/// The state profile for position, velocity, acceleration and jerk for a single DoF
FUNCTION_BLOCK Profile
VAR_INPUT
  limits : ProfileLimitsEnum;
  direction : ProfileDirectionEnum;
  jerkSigns : ProfileJerkSignsEnum;
  
  t, t_sum, j : ARRAY[0..6] OF LREAL;
  a, v, p : ARRAY[0..7] OF LREAL;

  pf, vf, af : LREAL; // Target (final) kinematic state
  
  hasBrake : BOOL;
  t_brake : LREAL; // Total time of the braking segments
  t_brakes, j_brakes, a_brakes, v_brakes, p_brakes : ARRAY[0..1] OF LREAL; // Allow up to two segments of braking before the "correct" profile starts 

END_VAR
VAR CONSTANT
  eps : LREAL := 1E-8;  
  infinity : LREAL := 1.7976931348623157E+308;
END_VAR
VAR_STAT
  root : Roots;
END_VAR

METHOD check : BOOL
VAR_INPUT
  jerkSigns : ProfileJerkSignsEnum;    
  limits : ProfileLimitsEnum;
  tf : LREAL;
  jf : LREAL;
  vMax : LREAL;
  vMin : LREAL;  
  aMax : LREAL;
  aMin : LREAL;
  jMax  : LREAL;
END_VAR
check := (ABS(jf) < ABS(jMax) + 1e-12) AND_THEN checkTime(jerkSigns, limits, tf, jf, vMax, vMin, aMax, aMin);
END_METHOD

/// For velocity interface
METHOD checkAcc : BOOL
VAR_INPUT
  jerkSigns : ProfileJerkSignsEnum;
  limits : ProfileLimitsEnum;  
  jf : LREAL;
  aMax : LREAL;
  aMin : LREAL;  
END_VAR
VAR
  i : INT;
  aUppLim : LREAL;
  aLowLim : LREAL;
END_VAR
IF (t[0] < 0)
THEN
  RETURN;
END_IF

t_sum[0] := t[0];
FOR i:=0 TO 5
DO
  IF (t[i+1] < 0)
  THEN
    RETURN;
  END_IF
  
  t_sum[i+1] := t_sum[i] + t[i+1];
END_FOR


IF limits = ProfileLimitsEnum.acc0
THEN
  IF t[1] < eps
  THEN
    RETURN;
  END_IF
END_IF


IF (t_sum[6] > 1E12) { // For numerical reasons, is that needed?}
THEN
  RETURN;        
END_IF

IF jerkSigns = ProfileJerkSignsEnum.uddu
THEN
  j[0] := jf;
  j[1] := 0;
  j[2] := -jf;
  j[3] := 0;
  j[4] := -jf;
  j[5] := 0;
  j[6] := jf;          
ELSE
  j[0] := jf;
  j[1] := 0;
  j[2] := -jf;
  j[3] := 0;
  j[4] := jf;
  j[5] := 0;
  j[6] := -jf;
END_IF


FOR i:=0 TO 6
DO
  a[i+1] := a[i] + t[i] * j[i];
  v[i+1] := v[i] + t[i] * (a[i] + t[i] * j[i] / 2);
  p[i+1] := p[i] + t[i] * (v[i] + t[i] * (a[i] / 2 + t[i] * j[i] / 6));        
END_FOR

      
THIS^.jerkSigns := jerkSigns;
THIS^.limits := limits;

aUppLim := SEL((aMax > 0), aMin, aMax) + 1E-12;
aLowLim := SEL((aMax > 0), aMax, aMin) - 1E-12;

// Velocity limit can be broken in the beginning if both initial velocity and acceleration are too high
checkAcc := ABS(v[7] - vf) < 1E-8
    AND_THEN ABS(a[7] - af) < 1E-12 // This is not really needed, but we want to double check
    AND_THEN a[1] >= aLowLim AND_THEN a[3] >= aLowLim AND_THEN a[5] >= aLowLim
    AND_THEN a[1] <= aUppLim AND_THEN a[3] <= aUppLim AND_THEN a[5] <= aUppLim;
END_METHOD

METHOD checkPositionExtremum : BOOL
VAR_INPUT
  t_ext, t_sum, t, p, v, a, j : LREAL;
END_VAR
VAR_IN_OUT
  ext : PositionExtremaStruct;     
END_VAR
VAR
  p_ext, v_Ext, a_ext : LREAL;
END_VAR
IF (0 < t_ext AND_THEN t_ext < t)
THEN
  integrate(t_ext, p, v, a, j, p:=p_ext, v:=v_ext, a:=a_ext);
  IF (a_ext > 0 AND_THEN p_ext < ext.minimum)
  THEN
    ext.minimum := p_ext;
    ext.t_min := t_sum + t_ext;
   ELSIF (a_ext < 0 AND_THEN p_ext > ext.maximum) 
   THEN
    ext.maximum := p_ext;
    ext.t_max := t_sum + t_ext; 
  END_IF
END_IF
END_METHOD

METHOD checkStepForPositionExtremum : BOOL
VAR_INPUT
  t_sum, t, p, v, a, j : LREAL;
END_VAR
VAR_IN_OUT
  ext : PositionExtremaStruct;  
END_VAR
VAR
  d, d_sqrt : LREAL;
END_VAR
IF (p < ext.minimum)
THEN 
  ext.minimum := p;
  ext.t_min := t_sum;
END_IF

IF (p > ext.maximum)
THEN 
  ext.maximum := p;
  ext.t_max := t_sum;
END_IF

IF (j <> 0) 
THEN
  d := a * a - 2 * j * v;
  IF (ABS(d) < eps)
  THEN
    checkPositionExtremum(-a / j, t_sum, t, p, v, a, j, ext:=ext);
   ELSIF (d > 0) 
   THEN
    d_sqrt := SQRT(d);
    checkPositionExtremum((-a - D_sqrt) / j, t_sum, t, p, v, a, j, ext:=ext);
    checkPositionExtremum((-a + D_sqrt) / j, t_sum, t, p, v, a, j, ext:=ext);           
  END_IF
END_IF
END_METHOD

METHOD checkTime : BOOL
VAR_INPUT
  jerkSigns : ProfileJerkSignsEnum;    
  limits : ProfileLimitsEnum;
  tf : LREAL;
  jf : LREAL;
  vMax : LREAL;
  vMin : LREAL;  
  aMax : LREAL;
  aMin : LREAL;  
END_VAR
// Time doesn't need to be checked as every profile has a: tf - ... equation
checkTime := checkVel(jerkSigns, limits, jf, vMax, vMin, aMax, aMin); // && (std::abs(t_sum[6] - tf) < 1e-8)
END_METHOD

/// For position interface
METHOD checkVel : BOOL
VAR_INPUT
  jerkSigns : ProfileJerkSignsEnum;    
  limits : ProfileLimitsEnum;
  jf : LREAL;
  vMax : LREAL;
  vMin : LREAL;  
  aMax : LREAL;
  aMin : LREAL;
END_VAR
VAR
  i : INT;
  v_a_zero : LREAL;
  vUppLim, vLowLim : LREAL;  
  aUppLim, aLowLim : LREAL;
END_VAR
IF (t[0] < 0) 
THEN
  RETURN;
END_IF

t_sum[0] := t[0];
FOR i:=0 TO 5
DO
  IF (t[i+1] < 0)
  THEN
    RETURN;
  END_IF
  
  t_sum[i+1] := t_sum[i] + t[i+1];  
END_FOR

IF limits = ProfileLimitsEnum.acc0_acc1_vel OR_ELSE limits = ProfileLimitsEnum.acc0_vel OR_ELSE limits = ProfileLimitsEnum.acc1_vel OR_ELSE limits = ProfileLimitsEnum.vel
THEN
  IF (t[3] < eps) 
  THEN
    RETURN;                    
  END_IF
END_IF

IF limits = ProfileLimitsEnum.acc0 OR_ELSE limits = ProfileLimitsEnum.acc0_acc1
THEN
  IF (t[1] < eps) 
  THEN
    RETURN;                    
  END_IF
END_IF

IF limits = ProfileLimitsEnum.acc1 OR_ELSE limits = ProfileLimitsEnum.acc0_acc1
THEN
  IF (t[5] < eps)
  THEN
    RETURN;            
  END_IF
END_IF

IF t_sum[6] > 1E12  // For numerical reasons, is that needed?
THEN
  RETURN;        
END_IF
        
IF jerkSigns = ProfileJerkSignsEnum.uddu
THEN
  j[0] := jf;
  j[1] := 0;
  j[2] := -jf;
  j[3] := 0;
  j[4] := -jf;
  j[5] := 0;
  j[6] := jf;
ELSE
  j[0] := jf;
  j[1] := 0;
  j[2] := -jf;
  j[3] := 0;
  j[4] := jf;
  j[5] := 0;
  j[6] := -jf;          
END_IF

vUppLim := SEL(vMax > 0, vMin, vMax) + 1E-12;
vLowLim := SEL(vMax > 0, vMax, vMin) - 1E-12;
        
FOR i:= 0 TO 6 
DO
  a[i+1] := a[i] + t[i] * j[i];
  v[i+1] := v[i] + t[i] * (a[i] + t[i] * j[i] / 2);
  p[i+1] := p[i] + t[i] * (v[i] + t[i] * (a[i] / 2 + t[i] * j[i] / 6));

  IF limits = ProfileLimitsEnum.acc0_acc1_vel OR_ELSE limits = ProfileLimitsEnum.acc0_vel OR_ELSE limits = ProfileLimitsEnum.acc1_vel OR_ELSE limits = ProfileLimitsEnum.vel
  THEN
    IF i = 2
    THEN
     a[3] := 0.0;
    END_IF
  END_IF 
  
  IF (i > 1 AND_THEN a[i+1] * a[i] < -eps) 
  THEN
    v_a_zero := v[i] - (a[i] * a[i]) / (2 * j[i]);
    IF (v_a_zero > vUppLim OR_ELSE v_a_zero < vLowLim)
    THEN
      RETURN;        
		END_IF
  END_IF
END_FOR


THIS^.jerkSigns := jerkSigns;
THIS^.limits := limits;

aUppLim := SEL((aMax > 0), aMin, aMax) + 1E-12;
aLowLim := SEL((aMax > 0), aMax, aMin) - 1E-12;

// Velocity limit can be broken in the beginning if both initial velocity and acceleration are too high
checkVel := ABS(p[7] - pf) < 1E-8
    AND_THEN ABS(v[7] - vf) < 1E-8
    AND_THEN ABS(a[7] - af) < 1E-10 // This is not really needed, but we want to double check
    // AND_THEN ABS(v[3]) <= vMaxAbs AND_THEN ABS(v[4]) <= vMaxAbs AND_THEN ABS(v[5]) <= vMaxAbs AND_THEN ABS(v[6]) <= vMaxAbs
    AND_THEN a[1] >= aLowLim AND_THEN a[3] >= aLowLim AND_THEN a[5] >= aLowLim
    AND_THEN a[1] <= aUppLim AND_THEN a[3] <= aUppLim AND_THEN a[5] <= aUppLim
    AND_THEN v[3] <= vUppLim AND_THEN v[4] <= vUppLim AND_THEN v[5] <= vUppLim AND_THEN v[6] <= vUppLim
    AND_THEN v[3] >= vLowLim AND_THEN v[4] >= vLowLim AND_THEN v[5] >= vLowLim AND_THEN v[6] >= vLowLim; // this is not really needed, but we want to double check
END_METHOD

METHOD firstStateAtPosition : BOOL
VAR_INPUT
  pt, offset : LREAL;
END_VAR
VAR_IN_OUT
  t_t, v_t, a_t : LREAL;
END_VAR
VAR
  i,h : INT;
  p_t : LREAL;
  polynom : ARRAY[0..4] OF LREAL;
END_VAR
FOR i:=0 TO 6
DO
  IF ABS(p[i] - pt) < eps
  THEN
    t_t := offset + SEL(i>0, 0, t_sum[i-1]);
    v_t := v[i];
    a_t := a[i];
    firstStateAtPosition := TRUE;
    RETURN;
	END_IF
  
  IF t[i] = 0
  THEN
    CONTINUE;
	END_IF
  
  polynom[0] := j[i]/6;
  polynom[1] := a[i]*0.5;
  polynom[2] := v[i];
  polynom[3] := p[i]-pt;
  root.solveCub(ADR(polynom));
  FOR h:=0 TO root.rootCount
  DO
    IF(0 < t[h] AND_THEN t[h] <= t[i])
    THEN
      t_t := offset + t[h] + SEL(i>0, 0, t_sum[i-1]);
      integrate(t[h], p[i], v[i], a[i], j[i], p_t, v_t, a_t);
      firstStateAtPosition := TRUE;
      RETURN;      
		END_IF
  END_FOR
  
END_FOR

IF ABS(pf-pt) < eps
THEN
  t_t := offset + t_sum[6];
  v_t := vf;
  a_t := af;
  firstStateAtPosition := TRUE;
  RETURN;      
END_IF
END_METHOD

 /// Integrate with constant jerk for duration t. Returns new position, new velocity, and new acceleration.
METHOD integrate
VAR_INPUT
  t, p0, v0, a0, j  : LREAL;
END_VAR
VAR_IN_OUT
  p, v, a : LREAL;
END_VAR
p := p0 + t * (v0 + t * (a0 * 0.5 + t * j / 6));
v := v0 + t * (a0 + t * j * 0.5);
a := a0 + t * j;
END_METHOD

METHOD positionExtrema : PositionExtremaStruct
VAR_INPUT
END_VAR
VAR
  i : INT;
  t_current_sum : LREAL;
END_VAR
positionExtrema.minimum := infinity;
positionExtrema.maximum := -infinity;

IF (hasBrake)
THEN
  IF (t_brakes[0] > 0.0)
  THEN
    checkStepForPositionExtremum(0.0, t_brakes[0], p_brakes[0], v_brakes[0], a_brakes[0], j_brakes[0], positionExtrema);
  
    IF (t_brakes[1] > 0.0) 
    THEN
      checkStepForPositionExtremum(t_brakes[0], t_brakes[1], p_brakes[1], v_brakes[1], a_brakes[1], j_brakes[1], positionExtrema);            
    END_IF
  END_IF
END_IF

t_current_sum := 0;        
FOR i:=0 TO 6
DO
  IF i > 0
  THEN
    t_current_sum := t_sum[i-1];
	END_IF
  
  checkStepForPositionExtremum(t_current_sum + t_brakes[i], t[i], p[i], v[i], a[i], j[i], positionExtrema);
END_FOR 

IF (pf < positionExtrema.minimum)
THEN
  positionExtrema.minimum := pf;
  positionExtrema.t_min := t_sum[6] + t_brakes[i];
END_IF 


IF (pf > positionExtrema.maximum) 
THEN
  positionExtrema.maximum := pf;
  positionExtrema.t_max := t_sum[6] + t_brakes[i];
END_IF
END_METHOD

/// Set boundary values for the position interface
METHOD setBoundaryPosition
VAR_INPUT
  p0_new, v0_new, a0_new, pf_new, vf_new, af_new : LREAL;
END_VAR
a[0] := a0_new;
v[0] := v0_new;
p[0] := p0_new;
af := af_new;
vf := vf_new;
pf := pf_new;
END_METHOD

/// Set boundary values for the velocity interface
METHOD setBoundaryVelocity
VAR_INPUT
  p0_new, v0_new, a0_new, vf_new, af_new : LREAL;
END_VAR
a[0] := a0_new;
v[0] := v0_new;
p[0] := p0_new;
af := af_new;
vf := vf_new;
END_METHOD

END_FUNCTION_BLOCK

(* stored: Version 1.1.0.1, ProductVersion 3.1.4024.9
   POU Profile: Id {1331731c-0677-4d13-b754-67c3077cc0c4}, SpecialFunc None
   Method check: Id {c707d6dc-e662-4300-aebc-c29e90e74532}
   Method checkAcc: Id {dec39d38-9a64-41bc-99b6-6a7b67c016da}
   Method checkPositionExtremum: Id {e3c5916b-156b-465a-87ae-6759453a325c}
   Method checkStepForPositionExtremum: Id {ce8df4c2-1570-4fbc-87ab-2de79032d446}
   Method checkTime: Id {a762f8df-7f20-4c45-819e-1ecbfa908ad5}
   Method checkVel: Id {1650deae-6774-4923-94a5-237877609b6a}
   Method firstStateAtPosition: Id {0159e4a6-0809-4a0c-b389-030aa446ea6f}
   Method integrate: Id {801ace88-741b-4b24-8760-4124fdd6b2b6}
   Method positionExtrema: Id {1a9ba528-afaf-4159-b889-acb983a16fac}
   Method setBoundaryPosition: Id {bcaf6cf3-3cdf-411e-b9b2-105283f26c0e}
   Method setBoundaryVelocity: Id {5e35273a-4554-4245-bfd9-f07367ed9a5c} *)
